{attribute 'qualified_only'}
VAR_GLOBAL
	sPistonEndStopMessages : STRING;
	bOn : BOOL;
	bAuto : BOOL;
	bStart : BOOL;
	bStop : BOOL;
	eMode : E_Mode;
END_VAR

(* stored: Version 1.1.0.1, ProductVersion 3.1.4024.9
   GVL HMI: Id {515f7d22-94cb-4f67-80c3-c968411175ad} *)
